// TIA Portal V18 export
TYPE "UDT_HCsDO"
// stored: IsFailsafeCompliant false
   STRUCT
      xHC3wvIncrease : Array[1..2] of Bool;
      xHC3wvDecrease : Array[1..2] of Bool;
      xHCPump1Cmd : Array[1..2] of Bool;
      xHCPump2Cmd : Array[1..2] of Bool;
   END_STRUCT;
END_TYPE
